// TIA Portal V17 export
// export: Created 2025-11-26T14:08:10.3197454Z, ExportSetting WithDefaults, WithReadOnly, DisplayName Totally Integrated Automation Portal, DisplayVersion V17 Update 7, DisplayName TIA Portal Openness, DisplayVersion V17 Update 7, DisplayName TIA Portal Version Control Interface, DisplayVersion V17, DisplayName SINAMICS Startdrive Advanced, DisplayVersion V17 SP2, DisplayName SINAMICS DCC, DisplayVersion V17 Update 1, DisplayName SINAMICS Startdrive G110M, G120, G120C, G120D, G120P, G115D, DisplayVersion V17 SP2, DisplayName SINAMICS Startdrive G130, G150, S120, S150, SINAMICS MV, S210, DisplayVersion V17 SP2, DisplayName STEP 7 Professional, DisplayVersion V17 Update 7, DisplayName STEP 7 Safety, DisplayVersion V17 Update 6, DisplayName WinCC Advanced, DisplayVersion V17 Update 7, DisplayName SIMATIC Visualization Architect, DisplayVersion V17 Update 7
DATA_BLOCK "[nome_robo]#FB_Rob_PN_A_DB"   // DB[numero_db]
{ S7_Optimized_Access := 'TRUE'; DB_Accessible_From_OPC_UA := 'FALSE' }
AUTHOR : VASS_V05
FAMILY : ROBPNA
VERSION : 0.0
// Ausgänge Roboter
// stored: AutoNumber false, CodeModifiedDate 2024-10-18T13:51:59.0675846Z, CompileDate 2024-11-07T14:09:47.9771046Z, CreationDate 2024-09-18T08:44:27.9878747Z, DBAccessibleFromOPCUA false, DBAccessibleFromWebserver true, DownloadWithoutReinit false, InstanceOfName FB_Rob_PN_A, InstanceOfNumber 201, InstanceOfType FB, InterfaceModifiedDate 2024-10-18T13:51:58.9948036Z, IsConsistent true, IsKnowHowProtected false, IsRetainMemResEnabled false, MemoryReserve 100, ModifiedDate 2024-11-12T16:05:11.9592259Z, ParameterModified 2024-04-29T15:32:09.0827443Z, StructureModified 2024-04-29T15:32:09.0827443Z, UDAEnableTagReadback false
"FB_Rob_PN_A"
   // VAR_INPUT
   //    Rob_A_F { ExternalAccessible := 'False'; ExternalVisible := 'False'; ExternalWritable := 'False'} : "ST_Rob_A_F";
   //    Rob_A { ExternalAccessible := 'False'; ExternalVisible := 'False'; ExternalWritable := 'False'} : "ST_Rob_A";
   //    Cfg : Word;
   // END_VAR
   // VAR_IN_OUT
   //    ST_ROB : "ST_Rob";
   // END_VAR
   // VAR
   //    diPOS_BLK { ExternalAccessible := 'False'; ExternalVisible := 'False'; ExternalWritable := 'False'} : DInt;
   //    "255" { ExternalAccessible := 'False'; ExternalVisible := 'False'; ExternalWritable := 'False'} : Bool;
   // END_VAR
BEGIN
END_DATA_BLOCK
